TYPE DeviceDataExt EXTENDS DeviceData :
STRUCT
	Justified: BOOL;
	ClingRequired: BOOL;
	ClingSize: cClingSize;
	CartonNum: DINT;
	CartonTracking: DINT;
	ToteRFID: DINT;
	ToteSide: DINT; //TODO, used for 1 or 2 phones in tote, to be removed
	JustifyNest: DINT;
END_STRUCT
END_TYPE

(* stored: Version 1.1.0.1, ProductVersion 3.1.4024.6
   DUT DeviceDataExt: Id {a9cda7fb-1b02-4b43-967b-6bf8cf8c75c2} *)
